FUNCTION F_AsciiNumberConvert : DINT
VAR_INPUT
	AsciiString : STRING;
END_VAR
VAR
	iValue: DINT;
	sValueString: STRING(255);
	sFirstNumber: STRING(255);
	sSecondNumber: STRING(255);
END_VAR


// Seperate number from string
sValueString := MID(AsciiString,4,4);
sFirstNumber := LEFT(sValueString,1);
sSecondNumber := LEFT(sValueString,2);
IF sFirstNumber = '0' AND sSecondNumber = '0' THEN
	iValue := STRING_TO_DINT(RIGHT(sValueString,2));
ELSIF sFirstNumber = '0' AND sSecondNumber <> '0' THEN
	iValue := STRING_TO_DINT(RIGHT(sValueString,3));
ELSE
	iValue := STRING_TO_DINT(sValueString);	
END_IF
F_AsciiNumberConvert := iValue;

END_FUNCTION

(* stored: Version 1.1.0.1, ProductVersion 3.1.4024.9
   POU F_AsciiNumberConvert: Id {74028c10-f7d1-461f-ba45-d589968c5dba}, SpecialFunc None *)
